{attribute 'qualified_only'}
VAR_GLOBAL RETAIN
	Actual_GLV_State :INT:=-1;
	Actual_In_State: INT:=-1;
	Actual_POs :REAL:=0;
END_VAR

(* stored: Version 1.1.0.1, ProductVersion 3.1.4024.4
   GVL QrRetVarState: Id {deda3d5a-8f3f-4362-950f-adbdb6a8e6cb} *)
